// TIA Portal V19 export
TYPE "LAF_typeMachineStatus"
TITLE = typeUnitStatus
// Information about the current unit status
// stored: Access Published
   STRUCT
      designSpeed : Real;   // provides the design speed of a machine (e.g. pcs/s)
      currentSpeed : Real;   // Provides the current speed of the machine (e.g. pcs/s)
      totalCounter : ULInt;   // Total counter of machine (good + defective counter)
      goodCounter : ULInt;   // Provides a counter for good parts
   END_STRUCT;
END_TYPE
